{attribute 'enable_dynamic_creation'}
FUNCTION_BLOCK FutureSleep EXTENDS FB_AbstructFuture
VAR_INPUT
END_VAR
VAR_OUTPUT
END_VAR
VAR
	_sleep_timer : TON;
	_sleep_time: TIME;
END_VAR

METHOD execute : BOOL // Return TRUE if finish.
_sleep_timer(IN := TRUE, PT := _sleep_time);
execute := _sleep_timer.Q;
END_METHOD

METHOD init : BOOL // Return TRUE if finish.
_sleep_timer(IN := FALSE);
init := TRUE;
END_METHOD

PROPERTY sleep_time : TIME
GET
sleep_time := _sleep_timer.ET;
END_GET
SET
_sleep_time := sleep_time;
END_SET
END_PROPERTY

END_FUNCTION_BLOCK

(* stored: Version 1.1.0.1, ProductVersion 3.1.4024.12
   POU FutureSleep: Id {8bbe7517-0dc1-4100-a111-c3897157da4f}, SpecialFunc None
   Method execute: Id {4b6e240c-c380-4850-b7b5-8246072f3874}
   Method init: Id {831745f4-91e6-4abd-9355-99a8e99d9e4c}
   Property sleep_time: Id {71da21e7-f780-46a0-ad0f-fb4e16fd8fdd}
   Get Get: Id {91ade5c2-e189-47d3-93a8-6aae32042fdd}
   Set Set: Id {d982e31a-7825-4a5f-8b8d-0f1de0afd6b4} *)
